(* Logix 5000 project; controller Sucrose_Main Emulate 5570 rev 20.12; software revision 20.01; part 19 of 30 *)
(* tags used below, declared in another part *)
   Alarm_ACK_Master_Timer : TIMER;
   Alarm_ACK_Sucrose : BOOL;
   DO_E22_7 : ALIAS FOR FLX_E22:7:O;   // Discrete Output EN2T_FLX 192.168.1.22
   FV920502_AOI : QSI_Flow_Valve;   // FV-92-05-02 FLT-23-05-02 VENT VALVE
   FV920601_AOI : QSI_Flow_Valve;   // FV-92-06-01 FLT-23-06-01 VENT VALVE
   FV920602_AOI : QSI_Flow_Valve;   // FV-92-06-02 FLT-23-06-02 VENT VALVE
   FV930401_AOI : QSI_Flow_Valve;   // FV-93-04-01 FLT-93-04-01 INLET VALVE
   FV930501_AOI : QSI_Flow_Valve;   // FV-93-05-01 PRE FILTER TRAIN 1 AIR BLOW INLET
   FV930502_AOI : QSI_Flow_Valve;   // FV-93-05-02 FINAL FILTER TRAIN 1 AIR BLOW VALVE
   FV930503_AOI : QSI_Flow_Valve;   // FV-93-05-03 INTEGRITY TEST TO SUPPLY TO FINAL FILTER TRAIN 1 VALVE
   FV930601_AOI : QSI_Flow_Valve;   // FV-93-06-01 PRE FILTER TRAIN 2 AIR BLOW INLET
   FV930602_AOI : QSI_Flow_Valve;   // FV-93-06-02 FINAL FILTER TRAIN 2 AIR BLOW OUTLET
   FV930603_AOI : QSI_Flow_Valve;   // FV-93-06-03 INTEGRITY TEST TO SUPPLY TO FINAL FILTER DRAIN VALVE
   FV930611_AOI : QSI_Flow_Valve;   // FV-93-06-11 PRE FILTER TRAIN 2 AIR BLOW OUTLET
   FV930612_AOI : QSI_Flow_Valve;   // FV-93-06-12 FINAL FILTER TRAIN 2 AIR BLOW OUTLET
   Messaging : Area_Ladder;
   Rung_Comment : BOOL;
   Sucrose_MM_Enable : BOOL;
   SucroseCIP_FILTRATION_REMOTE : CIP_REMOTE;
   SucroseDischarge : Area_Program;
   SucroseFiltration : Area_Program;
   SucroseReceiving : Area_Program;
   SucroseTanks : Area_Program;
(* FiltrationArea_EN2T_IO_Discrete_DO_E22_7, continued *)

ROUTINE _02_FV920502   (* ladder *)
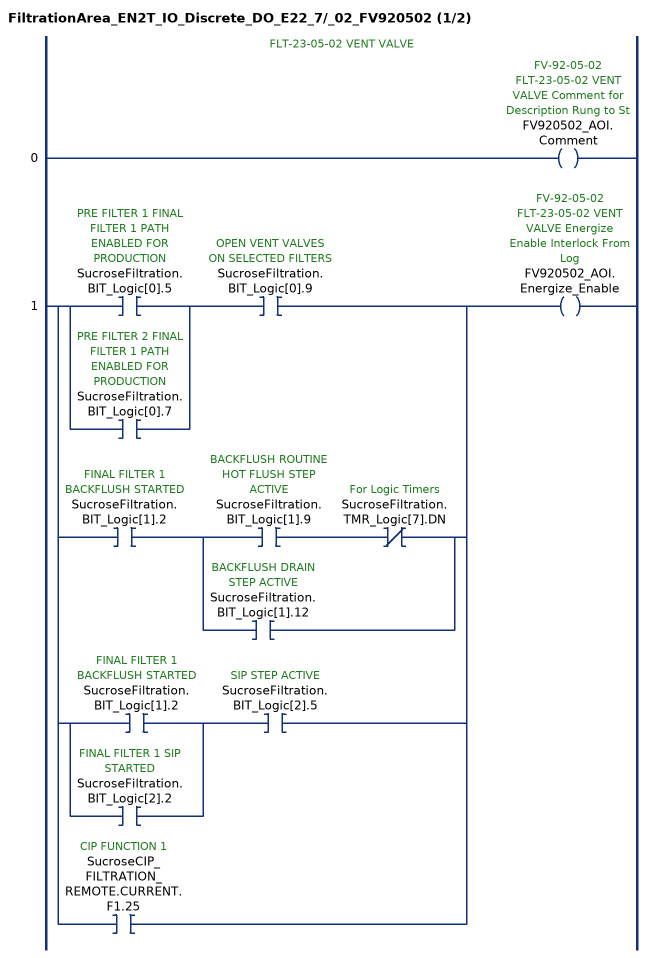
   // FLT-23-05-02 VENT VALVE
   0: OTE(FV920502_AOI.Comment);
   1: [[XIC(SucroseFiltration.BIT_Logic[0].5) ,XIC(SucroseFiltration.BIT_Logic[0].7) ] XIC(SucroseFiltration.BIT_Logic[0].9) ,XIC(SucroseFiltration.BIT_Logic[1].2) [XIC(SucroseFiltration.BIT_Logic[1].9) XIO(SucroseFiltration.TMR_Logic[7].DN) ,XIC(SucroseFiltration.BIT_Logic[1].12) ] ,[XIC(SucroseFiltration.BIT_Logic[1].2) ,XIC(SucroseFiltration.BIT_Logic[2].2) ] XIC(SucroseFiltration.BIT_Logic[2].5) ,XIC(SucroseCIP_FILTRATION_REMOTE.CURRENT.F1.25) ]OTE(FV920502_AOI.Energize_Enable);
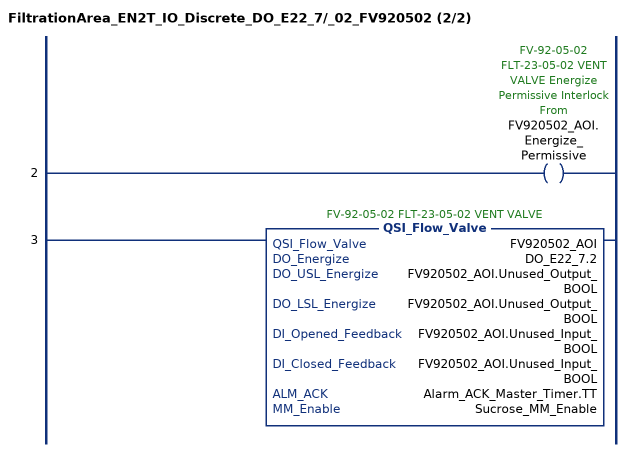
   2: OTE(FV920502_AOI.Energize_Permissive);
   3: QSI_Flow_Valve(FV920502_AOI,DO_E22_7.2,FV920502_AOI.Unused_Output_BOOL,FV920502_AOI.Unused_Output_BOOL,FV920502_AOI.Unused_Input_BOOL,FV920502_AOI.Unused_Input_BOOL,Alarm_ACK_Master_Timer.TT,Sucrose_MM_Enable);
END_ROUTINE

ROUTINE _03_FV920601   (* ladder *)
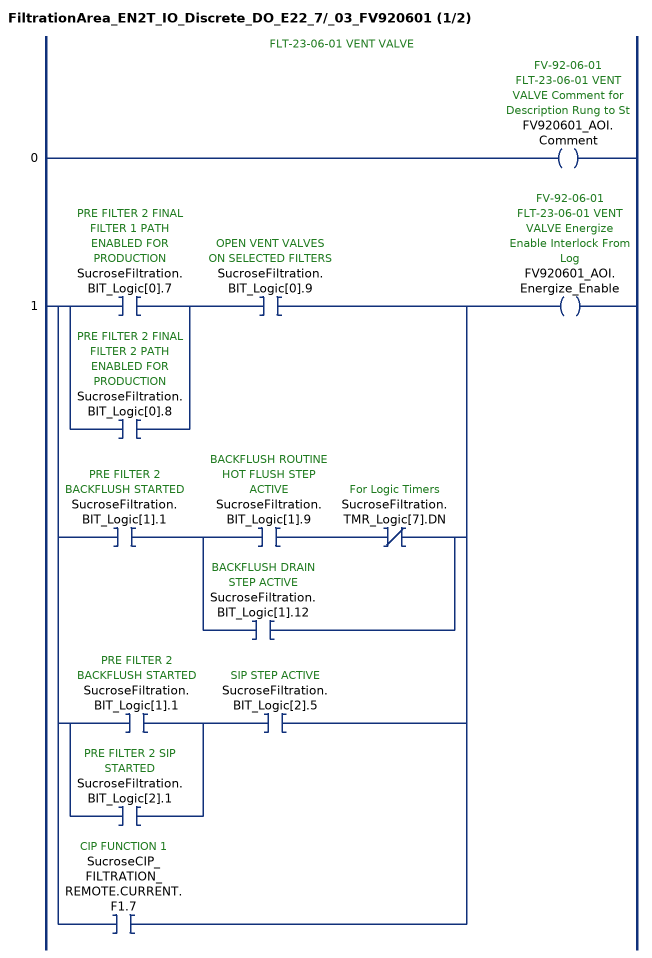
   // FLT-23-06-01 VENT VALVE
   0: OTE(FV920601_AOI.Comment);
   1: [[XIC(SucroseFiltration.BIT_Logic[0].7) ,XIC(SucroseFiltration.BIT_Logic[0].8) ] XIC(SucroseFiltration.BIT_Logic[0].9) ,XIC(SucroseFiltration.BIT_Logic[1].1) [XIC(SucroseFiltration.BIT_Logic[1].9) XIO(SucroseFiltration.TMR_Logic[7].DN) ,XIC(SucroseFiltration.BIT_Logic[1].12) ] ,[XIC(SucroseFiltration.BIT_Logic[1].1) ,XIC(SucroseFiltration.BIT_Logic[2].1) ] XIC(SucroseFiltration.BIT_Logic[2].5) ,XIC(SucroseCIP_FILTRATION_REMOTE.CURRENT.F1.7) ]OTE(FV920601_AOI.Energize_Enable);
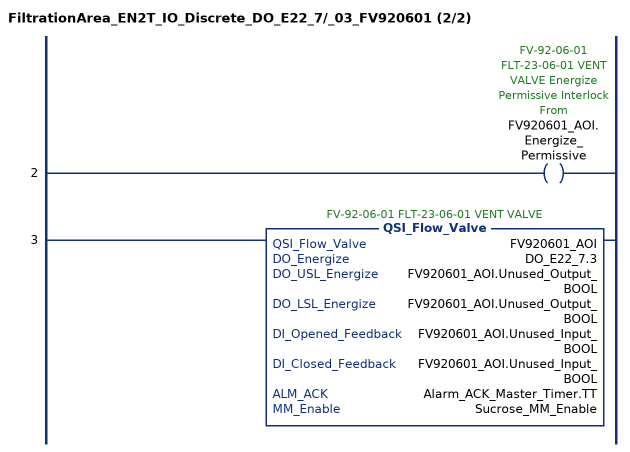
   2: OTE(FV920601_AOI.Energize_Permissive);
   3: QSI_Flow_Valve(FV920601_AOI,DO_E22_7.3,FV920601_AOI.Unused_Output_BOOL,FV920601_AOI.Unused_Output_BOOL,FV920601_AOI.Unused_Input_BOOL,FV920601_AOI.Unused_Input_BOOL,Alarm_ACK_Master_Timer.TT,Sucrose_MM_Enable);
END_ROUTINE

ROUTINE _04_FV930401   (* ladder *)
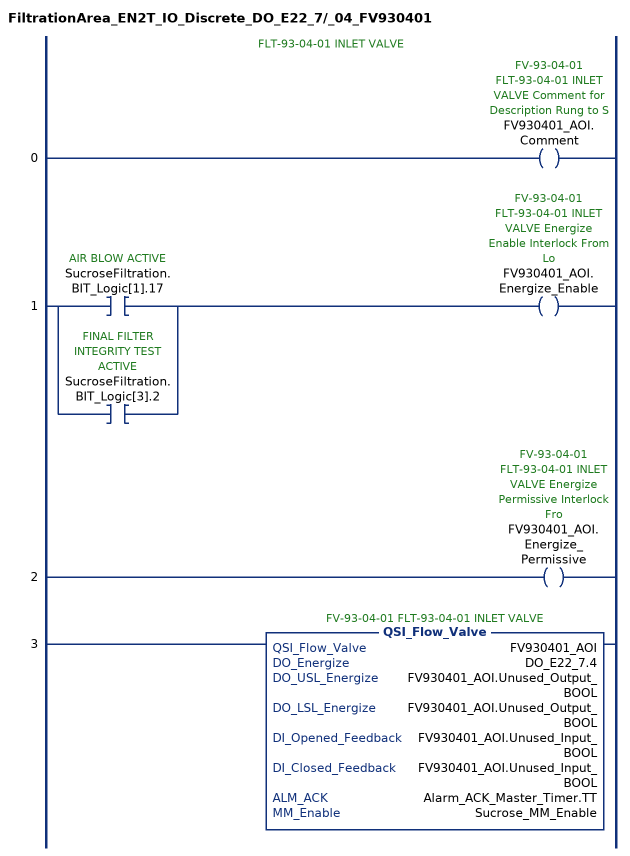
   // FLT-93-04-01 INLET VALVE
   0: OTE(FV930401_AOI.Comment);
   1: [XIC(SucroseFiltration.BIT_Logic[1].17) ,XIC(SucroseFiltration.BIT_Logic[3].2) ]OTE(FV930401_AOI.Energize_Enable);
   2: OTE(FV930401_AOI.Energize_Permissive);
   3: QSI_Flow_Valve(FV930401_AOI,DO_E22_7.4,FV930401_AOI.Unused_Output_BOOL,FV930401_AOI.Unused_Output_BOOL,FV930401_AOI.Unused_Input_BOOL,FV930401_AOI.Unused_Input_BOOL,Alarm_ACK_Master_Timer.TT,Sucrose_MM_Enable);
END_ROUTINE

ROUTINE _05_FV930501   (* ladder *)
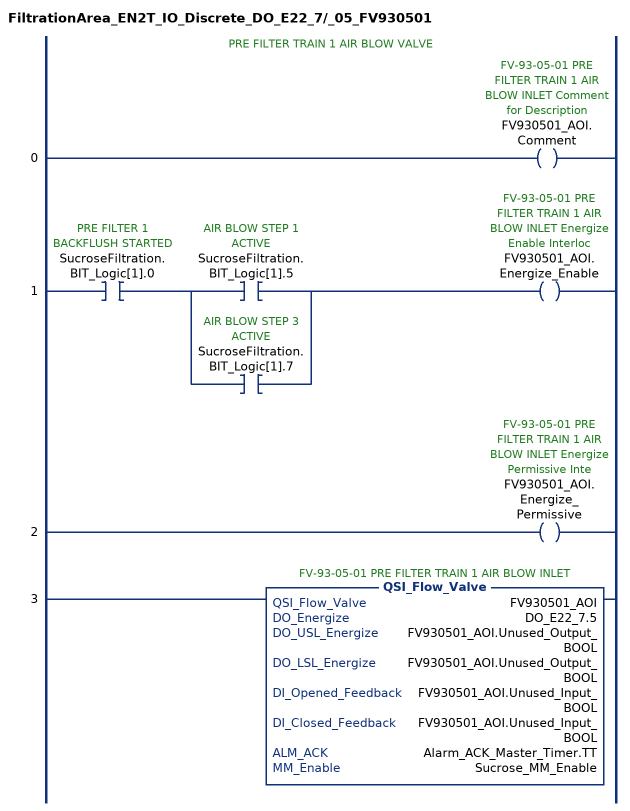
   // PRE FILTER TRAIN 1 AIR BLOW VALVE
   0: OTE(FV930501_AOI.Comment);
   1: XIC(SucroseFiltration.BIT_Logic[1].0)[XIC(SucroseFiltration.BIT_Logic[1].5) ,XIC(SucroseFiltration.BIT_Logic[1].7) ]OTE(FV930501_AOI.Energize_Enable);
   2: OTE(FV930501_AOI.Energize_Permissive);
   3: QSI_Flow_Valve(FV930501_AOI,DO_E22_7.5,FV930501_AOI.Unused_Output_BOOL,FV930501_AOI.Unused_Output_BOOL,FV930501_AOI.Unused_Input_BOOL,FV930501_AOI.Unused_Input_BOOL,Alarm_ACK_Master_Timer.TT,Sucrose_MM_Enable);
END_ROUTINE

ROUTINE _06_FV930503   (* ladder *)
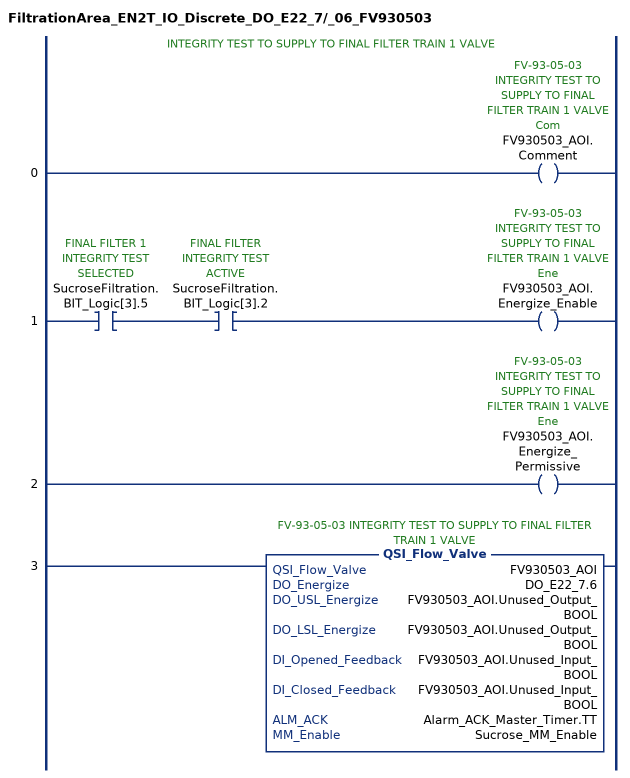
   // INTEGRITY TEST TO SUPPLY TO FINAL FILTER TRAIN 1 VALVE
   0: OTE(FV930503_AOI.Comment);
   1: XIC(SucroseFiltration.BIT_Logic[3].5)XIC(SucroseFiltration.BIT_Logic[3].2)OTE(FV930503_AOI.Energize_Enable);
   2: OTE(FV930503_AOI.Energize_Permissive);
   3: QSI_Flow_Valve(FV930503_AOI,DO_E22_7.6,FV930503_AOI.Unused_Output_BOOL,FV930503_AOI.Unused_Output_BOOL,FV930503_AOI.Unused_Input_BOOL,FV930503_AOI.Unused_Input_BOOL,Alarm_ACK_Master_Timer.TT,Sucrose_MM_Enable);
END_ROUTINE

ROUTINE _07_FV930502   (* ladder *)
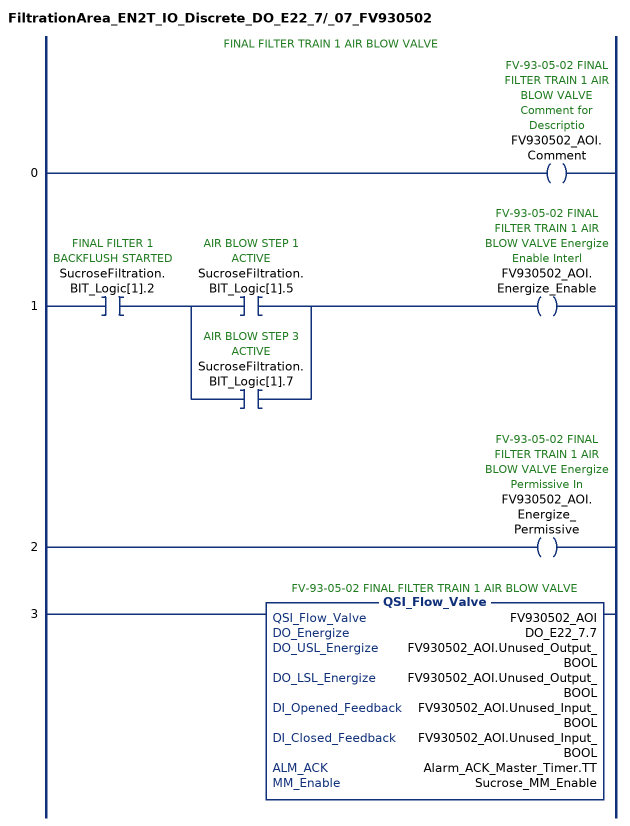
   // FINAL FILTER TRAIN 1 AIR BLOW VALVE
   0: OTE(FV930502_AOI.Comment);
   1: XIC(SucroseFiltration.BIT_Logic[1].2)[XIC(SucroseFiltration.BIT_Logic[1].5) ,XIC(SucroseFiltration.BIT_Logic[1].7) ]OTE(FV930502_AOI.Energize_Enable);
   2: OTE(FV930502_AOI.Energize_Permissive);
   3: QSI_Flow_Valve(FV930502_AOI,DO_E22_7.7,FV930502_AOI.Unused_Output_BOOL,FV930502_AOI.Unused_Output_BOOL,FV930502_AOI.Unused_Input_BOOL,FV930502_AOI.Unused_Input_BOOL,Alarm_ACK_Master_Timer.TT,Sucrose_MM_Enable);
END_ROUTINE

ROUTINE _08_FV930601   (* ladder *)
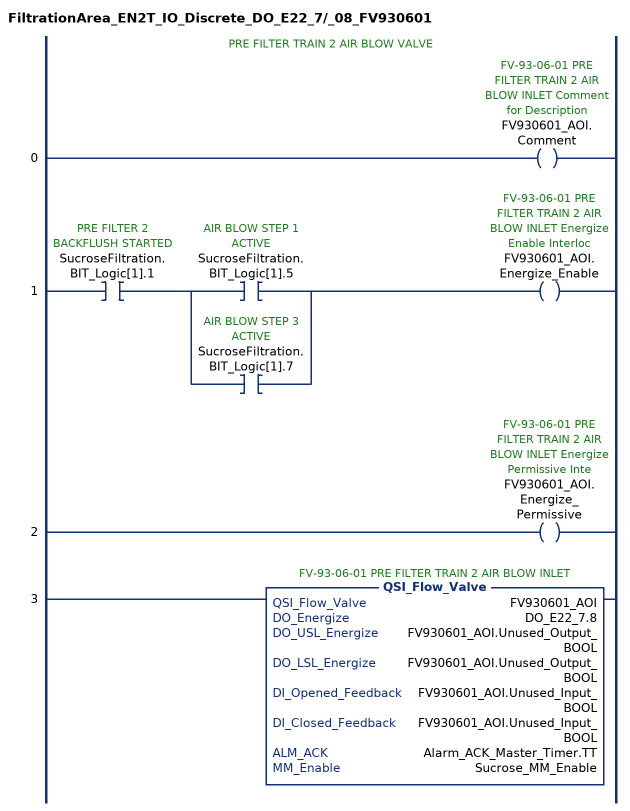
   // PRE FILTER TRAIN 2 AIR BLOW VALVE
   0: OTE(FV930601_AOI.Comment);
   1: XIC(SucroseFiltration.BIT_Logic[1].1)[XIC(SucroseFiltration.BIT_Logic[1].5) ,XIC(SucroseFiltration.BIT_Logic[1].7) ]OTE(FV930601_AOI.Energize_Enable);
   2: OTE(FV930601_AOI.Energize_Permissive);
   3: QSI_Flow_Valve(FV930601_AOI,DO_E22_7.8,FV930601_AOI.Unused_Output_BOOL,FV930601_AOI.Unused_Output_BOOL,FV930601_AOI.Unused_Input_BOOL,FV930601_AOI.Unused_Input_BOOL,Alarm_ACK_Master_Timer.TT,Sucrose_MM_Enable);
END_ROUTINE

ROUTINE _09_FV920602   (* ladder *)
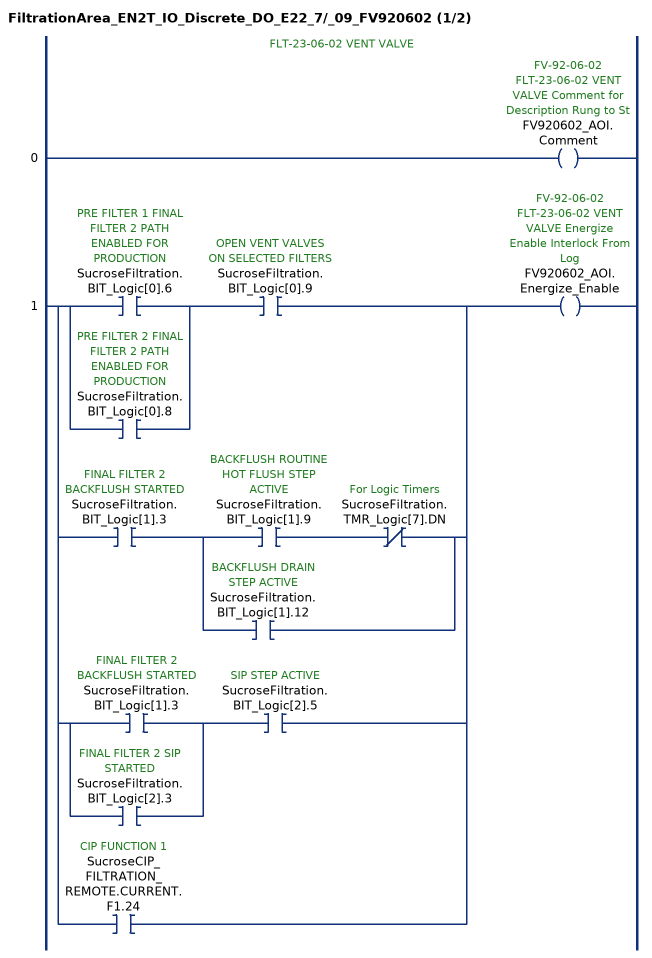
   // FLT-23-06-02 VENT VALVE
   0: OTE(FV920602_AOI.Comment);
   1: [[XIC(SucroseFiltration.BIT_Logic[0].6) ,XIC(SucroseFiltration.BIT_Logic[0].8) ] XIC(SucroseFiltration.BIT_Logic[0].9) ,XIC(SucroseFiltration.BIT_Logic[1].3) [XIC(SucroseFiltration.BIT_Logic[1].9) XIO(SucroseFiltration.TMR_Logic[7].DN) ,XIC(SucroseFiltration.BIT_Logic[1].12) ] ,[XIC(SucroseFiltration.BIT_Logic[1].3) ,XIC(SucroseFiltration.BIT_Logic[2].3) ] XIC(SucroseFiltration.BIT_Logic[2].5) ,XIC(SucroseCIP_FILTRATION_REMOTE.CURRENT.F1.24) ]OTE(FV920602_AOI.Energize_Enable);
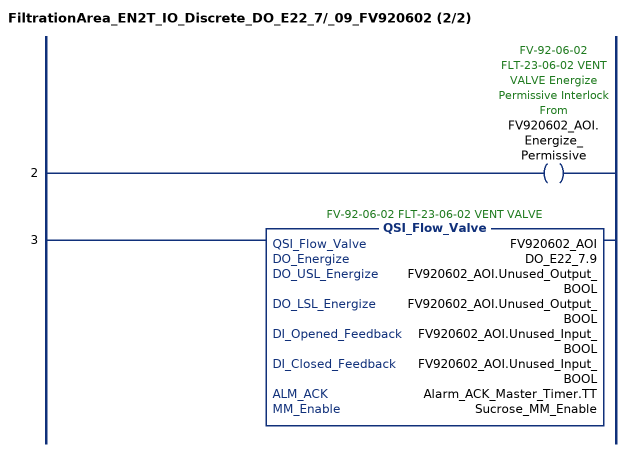
   2: OTE(FV920602_AOI.Energize_Permissive);
   3: QSI_Flow_Valve(FV920602_AOI,DO_E22_7.9,FV920602_AOI.Unused_Output_BOOL,FV920602_AOI.Unused_Output_BOOL,FV920602_AOI.Unused_Input_BOOL,FV920602_AOI.Unused_Input_BOOL,Alarm_ACK_Master_Timer.TT,Sucrose_MM_Enable);
END_ROUTINE

ROUTINE _10_FV930603   (* ladder *)
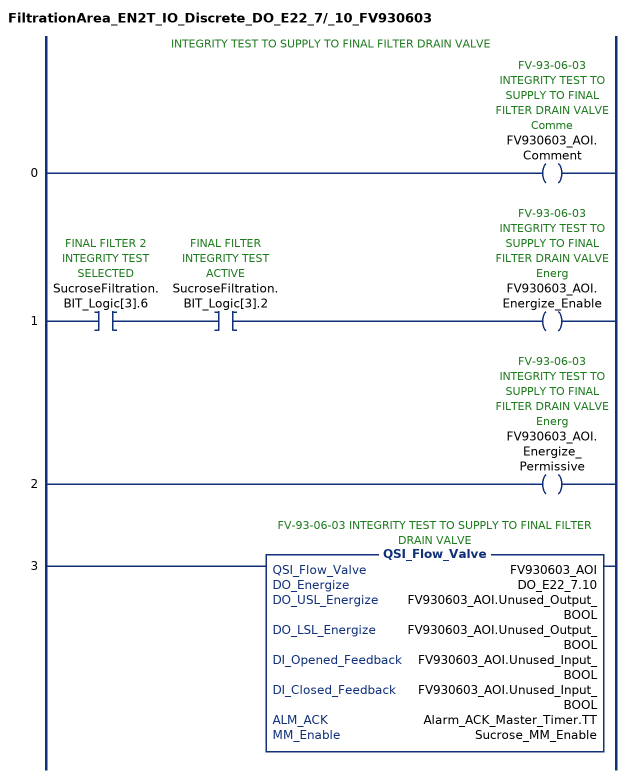
   // INTEGRITY TEST TO SUPPLY TO FINAL FILTER DRAIN VALVE
   0: OTE(FV930603_AOI.Comment);
   1: XIC(SucroseFiltration.BIT_Logic[3].6)XIC(SucroseFiltration.BIT_Logic[3].2)OTE(FV930603_AOI.Energize_Enable);
   2: OTE(FV930603_AOI.Energize_Permissive);
   3: QSI_Flow_Valve(FV930603_AOI,DO_E22_7.10,FV930603_AOI.Unused_Output_BOOL,FV930603_AOI.Unused_Output_BOOL,FV930603_AOI.Unused_Input_BOOL,FV930603_AOI.Unused_Input_BOOL,Alarm_ACK_Master_Timer.TT,Sucrose_MM_Enable);
END_ROUTINE

ROUTINE _11_FV930602   (* ladder *)
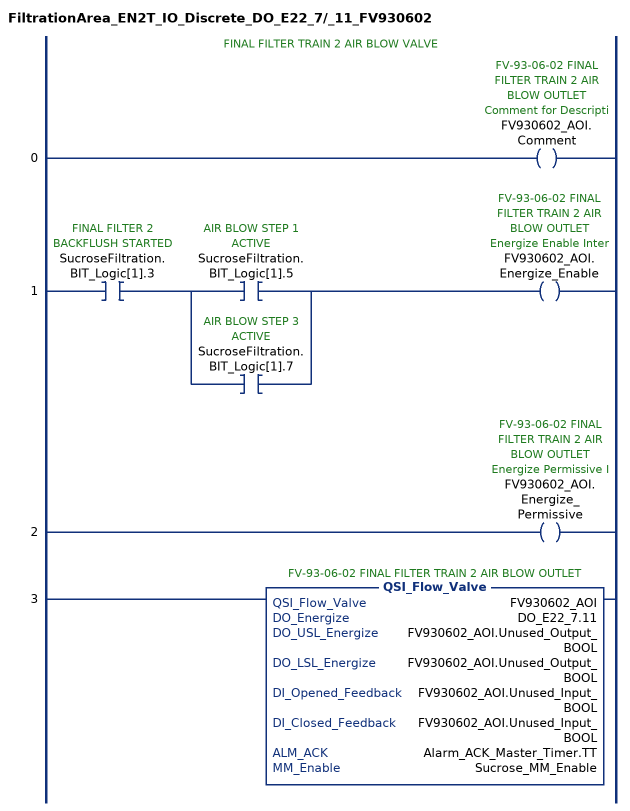
   // FINAL FILTER TRAIN 2 AIR BLOW VALVE
   0: OTE(FV930602_AOI.Comment);
   1: XIC(SucroseFiltration.BIT_Logic[1].3)[XIC(SucroseFiltration.BIT_Logic[1].5) ,XIC(SucroseFiltration.BIT_Logic[1].7) ]OTE(FV930602_AOI.Energize_Enable);
   2: OTE(FV930602_AOI.Energize_Permissive);
   3: QSI_Flow_Valve(FV930602_AOI,DO_E22_7.11,FV930602_AOI.Unused_Output_BOOL,FV930602_AOI.Unused_Output_BOOL,FV930602_AOI.Unused_Input_BOOL,FV930602_AOI.Unused_Input_BOOL,Alarm_ACK_Master_Timer.TT,Sucrose_MM_Enable);
END_ROUTINE

ROUTINE _12_FV930611   (* ladder *)
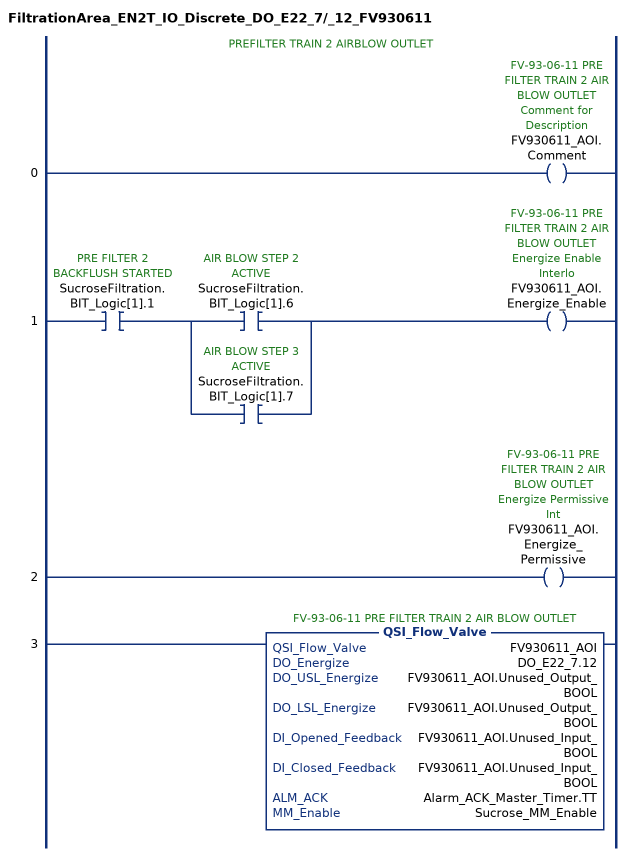
   // PREFILTER TRAIN 2 AIRBLOW OUTLET
   0: OTE(FV930611_AOI.Comment);
   1: XIC(SucroseFiltration.BIT_Logic[1].1)[XIC(SucroseFiltration.BIT_Logic[1].6) ,XIC(SucroseFiltration.BIT_Logic[1].7) ]OTE(FV930611_AOI.Energize_Enable);
   2: OTE(FV930611_AOI.Energize_Permissive);
   3: QSI_Flow_Valve(FV930611_AOI,DO_E22_7.12,FV930611_AOI.Unused_Output_BOOL,FV930611_AOI.Unused_Output_BOOL,FV930611_AOI.Unused_Input_BOOL,FV930611_AOI.Unused_Input_BOOL,Alarm_ACK_Master_Timer.TT,Sucrose_MM_Enable);
END_ROUTINE

ROUTINE _13_FV930612   (* ladder *)
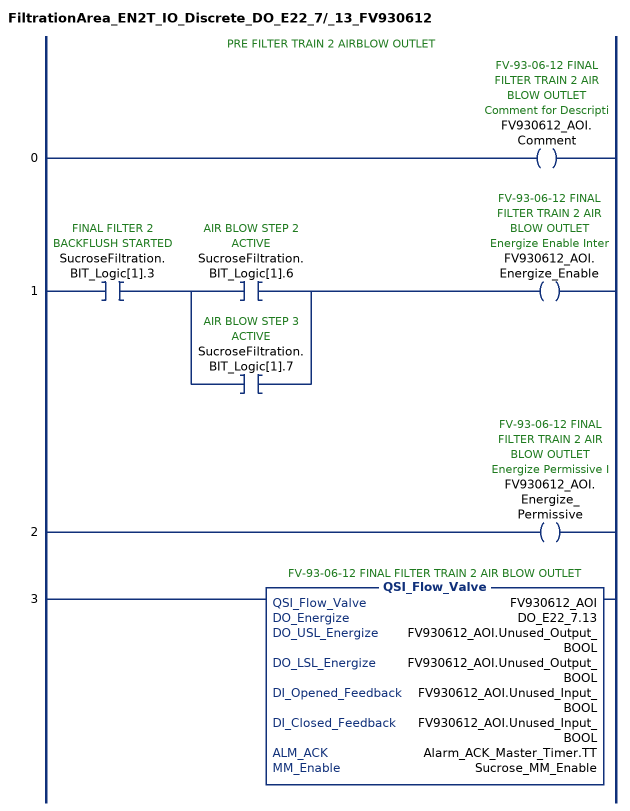
   // PRE FILTER TRAIN 2 AIRBLOW OUTLET
   0: OTE(FV930612_AOI.Comment);
   1: XIC(SucroseFiltration.BIT_Logic[1].3)[XIC(SucroseFiltration.BIT_Logic[1].6) ,XIC(SucroseFiltration.BIT_Logic[1].7) ]OTE(FV930612_AOI.Energize_Enable);
   2: OTE(FV930612_AOI.Energize_Permissive);
   3: QSI_Flow_Valve(FV930612_AOI,DO_E22_7.13,FV930612_AOI.Unused_Output_BOOL,FV930612_AOI.Unused_Output_BOOL,FV930612_AOI.Unused_Input_BOOL,FV930612_AOI.Unused_Input_BOOL,Alarm_ACK_Master_Timer.TT,Sucrose_MM_Enable);
END_ROUTINE

ROUTINE MainRoutine   (* ladder *)
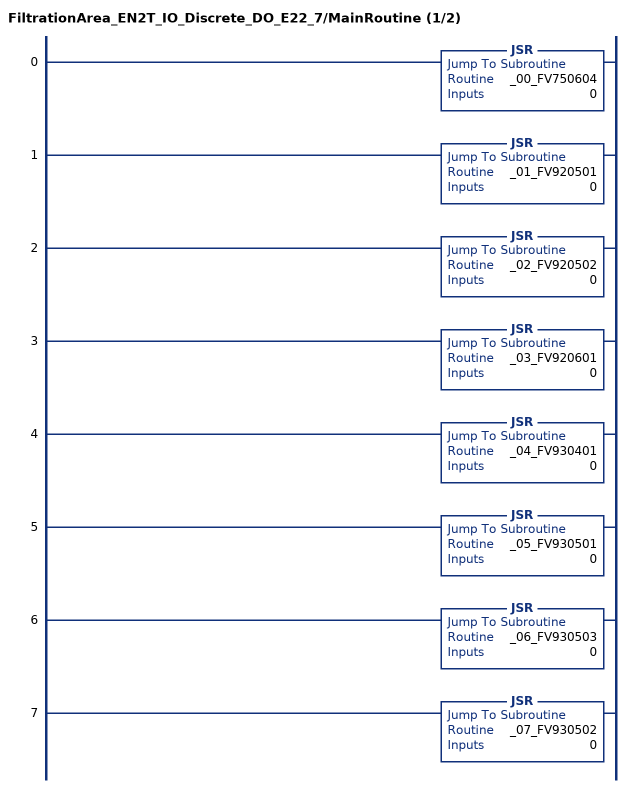
   0: JSR(_00_FV750604,0);
   1: JSR(_01_FV920501,0);
   2: JSR(_02_FV920502,0);
   3: JSR(_03_FV920601,0);
   4: JSR(_04_FV930401,0);
   5: JSR(_05_FV930501,0);
   6: JSR(_06_FV930503,0);
   7: JSR(_07_FV930502,0);
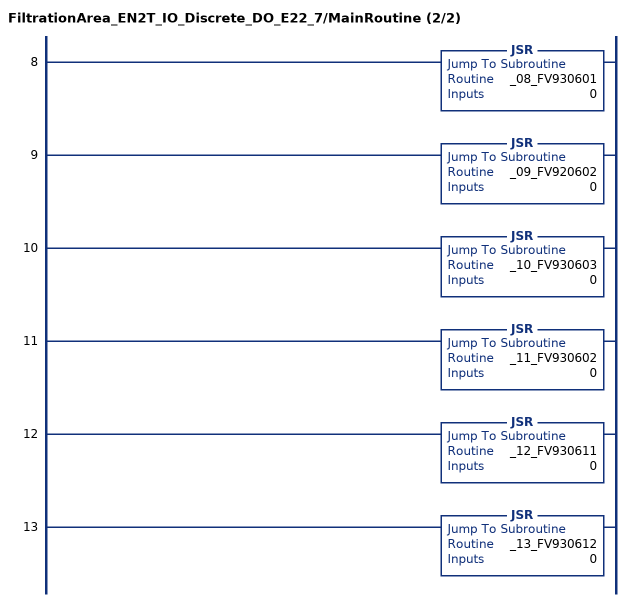
   8: JSR(_08_FV930601,0);
   9: JSR(_09_FV920602,0);
   10: JSR(_10_FV930603,0);
   11: JSR(_11_FV930602,0);
   12: JSR(_12_FV930611,0);
   13: JSR(_13_FV930612,0);
END_ROUTINE
END_PROGRAM

PROGRAM Master_Main   (* main routine MainRoutine *)

ROUTINE Alarm_ACK   (* ladder *)
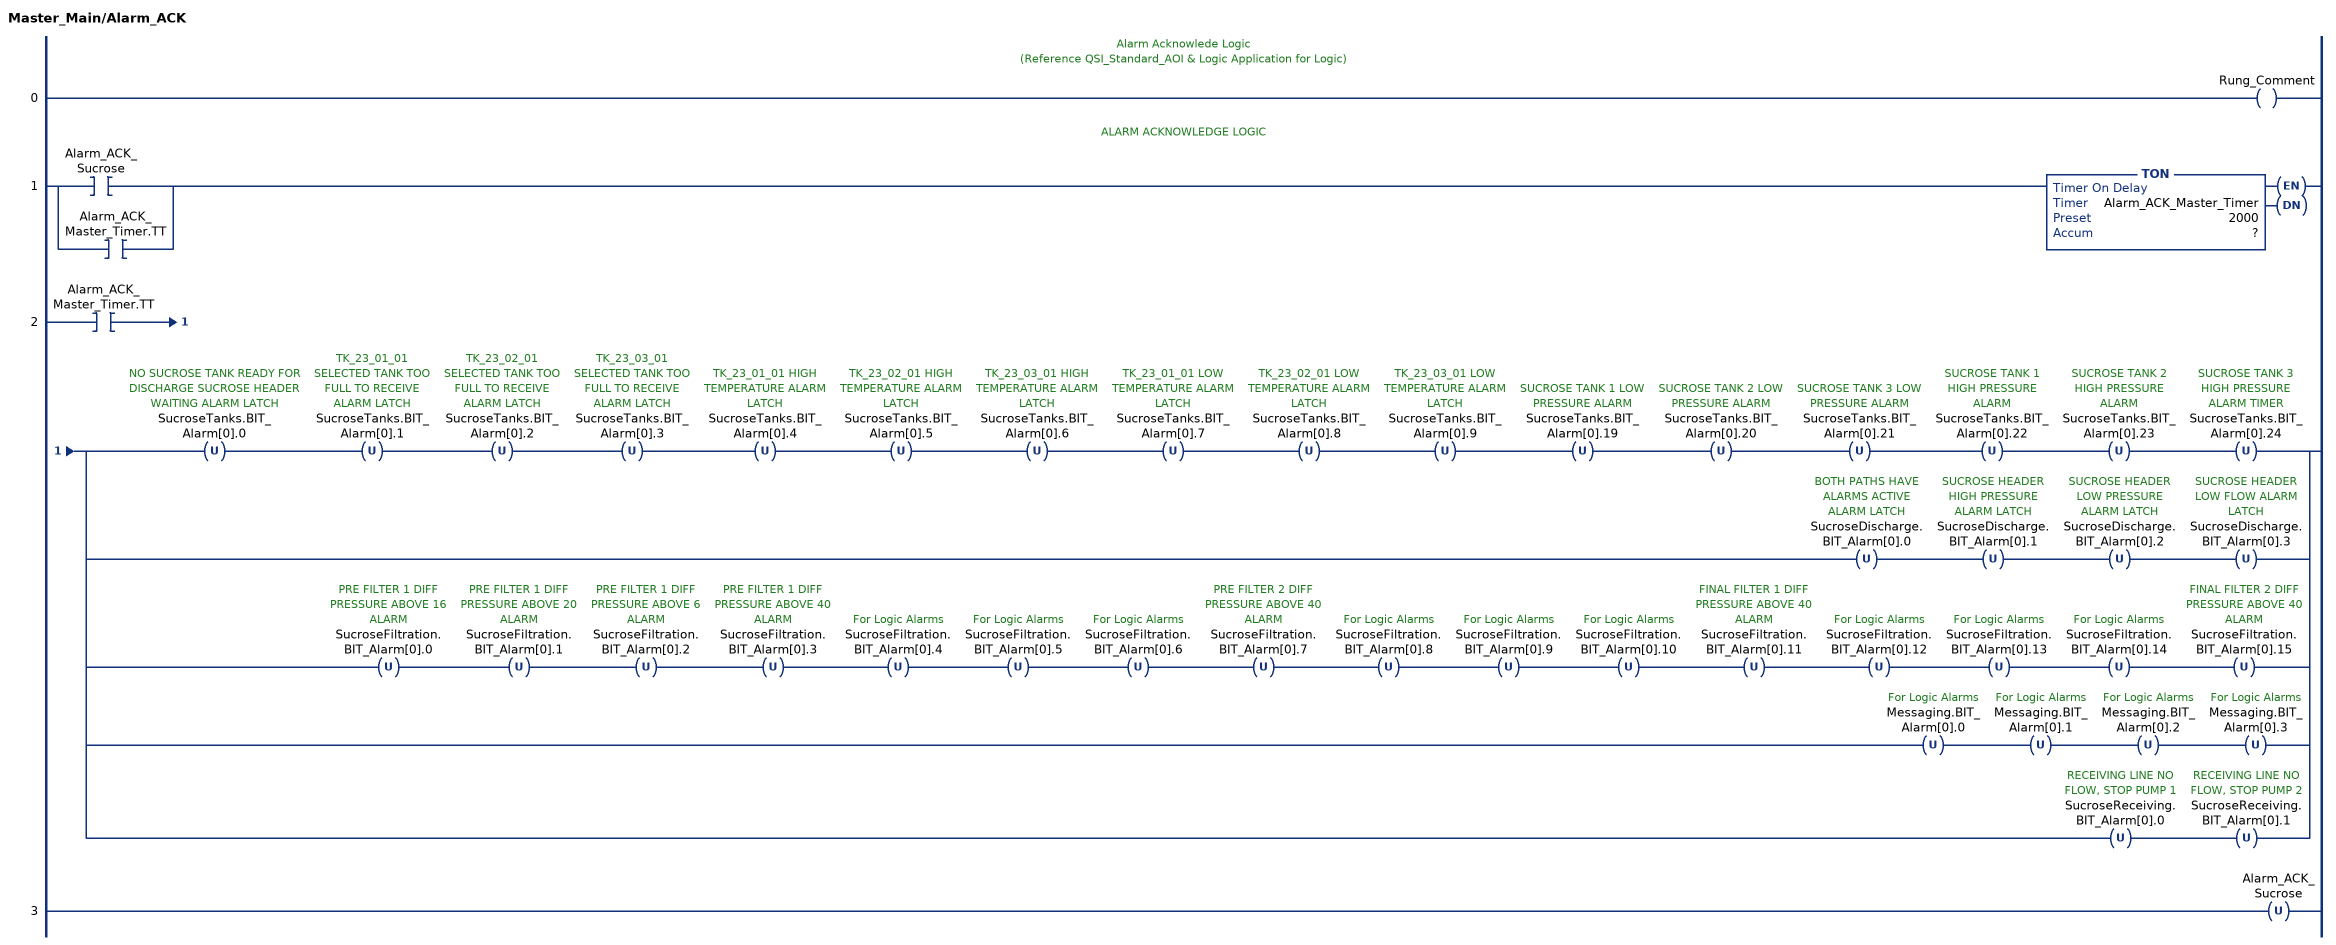
   // Alarm Acknowlede Logic
   // (Reference QSI_Standard_AOI & Logic Application for Logic)
   0: OTE(Rung_Comment);
   // ALARM ACKNOWLEDGE LOGIC
   1: [XIC(Alarm_ACK_Sucrose) ,XIC(Alarm_ACK_Master_Timer.TT) ]TON(Alarm_ACK_Master_Timer,?,?);
   2: XIC(Alarm_ACK_Master_Timer.TT)[OTU(SucroseTanks.BIT_Alarm[0].0) OTU(SucroseTanks.BIT_Alarm[0].1) OTU(SucroseTanks.BIT_Alarm[0].2) OTU(SucroseTanks.BIT_Alarm[0].3) OTU(SucroseTanks.BIT_Alarm[0].4) OTU(SucroseTanks.BIT_Alarm[0].5) OTU(SucroseTanks.BIT_Alarm[0].6) OTU(SucroseTanks.BIT_Alarm[0].7) OTU(SucroseTanks.BIT_Alarm[0].8) OTU(SucroseTanks.BIT_Alarm[0].9) OTU(SucroseTanks.BIT_Alarm[0].19) OTU(SucroseTanks.BIT_Alarm[0].20) OTU(SucroseTanks.BIT_Alarm[0].21) OTU(SucroseTanks.BIT_Alarm[0].22) OTU(SucroseTanks.BIT_Alarm[0].23) OTU(SucroseTanks.BIT_Alarm[0].24) ,OTU(SucroseDischarge.BIT_Alarm[0].0) OTU(SucroseDischarge.BIT_Alarm[0].1) OTU(SucroseDischarge.BIT_Alarm[0].2) OTU(SucroseDischarge.BIT_Alarm[0].3) ,OTU(SucroseFiltration.BIT_Alarm[0].0) OTU(SucroseFiltration.BIT_Alarm[0].1) OTU(SucroseFiltration.BIT_Alarm[0].2) OTU(SucroseFiltration.BIT_Alarm[0].3) OTU(SucroseFiltration.BIT_Alarm[0].4) OTU(SucroseFiltration.BIT_Alarm[0].5) OTU(SucroseFiltration.BIT_Alarm[0].6) OTU(SucroseFiltration.BIT_Alarm[0].7) OTU(SucroseFiltration.BIT_Alarm[0].8) OTU(SucroseFiltration.BIT_Alarm[0].9) OTU(SucroseFiltration.BIT_Alarm[0].10) OTU(SucroseFiltration.BIT_Alarm[0].11) OTU(SucroseFiltration.BIT_Alarm[0].12) OTU(SucroseFiltration.BIT_Alarm[0].13) OTU(SucroseFiltration.BIT_Alarm[0].14) OTU(SucroseFiltration.BIT_Alarm[0].15) ,OTU(Messaging.BIT_Alarm[0].0) OTU(Messaging.BIT_Alarm[0].1) OTU(Messaging.BIT_Alarm[0].2) OTU(Messaging.BIT_Alarm[0].3) ,OTU(SucroseReceiving.BIT_Alarm[0].0) OTU(SucroseReceiving.BIT_Alarm[0].1) ];
   3: OTU(Alarm_ACK_Sucrose);
END_ROUTINE
